PROGRAM A_Program
VAR
END_VAR

B_Program();

END_PROGRAM

(* stored: Version 1.1.0.1, ProductVersion 3.1.4025.12
   POU A_Program: Id {f11a5492-28ad-409b-8a88-13c6a15fc4ad}, SpecialFunc None *)
